// TIA Portal V18 export
VAR_GLOBAL   // PLC tag table "Lifting"
END_VAR
VAR_GLOBAL CONSTANT   // user constants
   Job_Run_in : Int := 10;   // 进料任务分配中
   Job_Run_out : Int := 15;   // 出料任务分配中
   Job_Run : Int := 60;   // 有任务在提升机运行
   Job_Run_in_done : Int := 11;   // 进料任务完成
   Job_Run_out_done : Int := 16;   // 出料任务完成
   Liftinghavepart : Int := 66;   // 提升机有托盘
END_VAR
